// TIA Portal V18 export
TYPE "MEStoPLC_ST350_ext"
// stored: IsFailsafeCompliant false
   STRUCT
      MainCheckIn { S7_SetPoint := 'True'} : "MEStoPLC_MainCheckIn_ext";   // MES反馈主件查询结果
      SubCheckIn { S7_SetPoint := 'True'} : "MEStoPLC_SubCheckIn_ext";   // MES反馈子件查询结果
      ScanResultsStored { S7_SetPoint := 'True'} : "MEStoPLC_ResultsStoredScanExchange_ext";   // 手持扫码枪上料查询事件反馈
      MarkingPrintExchange { S7_SetPoint := 'True'} : "MEStoPLC_PrintExchange_ext";   // MES反馈打印数据
      MainCheckOut { S7_SetPoint := 'True'} : "MEStoPLC_MainCheckOut_ext";   // MES反馈Processing记录结果
      Common { S7_SetPoint := 'True'} : "MEStoPLC_Common_ext";   // MES反馈公共区
   END_STRUCT;
END_TYPE
